// TIA Portal V18 export
FUNCTION_BLOCK "Conveyor"   // FB2, FBD
{ S7_Optimized_Access := 'TRUE' }
VERSION : 0.1
// stored: AutoNumber true, IsIECCheckEnabled true, IsRetainMemResEnabled false, MemoryReserve 100, SetENOAutomatically false, UDAEnableTagReadback false
   VAR_INPUT
      automaticMode : Bool;
      manualMode : Bool;
      jogRight : Bool;
      run : Bool;
   END_VAR
   VAR_OUTPUT
      conveyorRight : Bool;
      conveyorLeft : Bool;
   END_VAR
   VAR
      statRequest : Bool;
      statRelease : Bool;
   END_VAR
BEGIN

REGION Network 1 (SCL)
   //=============================================================================
   //Siemens AG // (c)Copyright (2018)
   //-----------------------------------------------------------------------------
   // Library: -
   // Tested with: CPU 1517-3 PN/DP V2.5
   // Engineering: TIA Portal V15
   // Restrictions: -
   // Requirements: PLC (S7-1500)
   // Functionality: Conveyor
   //-----------------------------------------------------------------------------
   // Change log table:
   // Version  Date      Expert in charge  Changes applied
   // 01.00.00 24.08.18  Siemens           First released version
   //=============================================================================
END_REGION

REGION Network 2
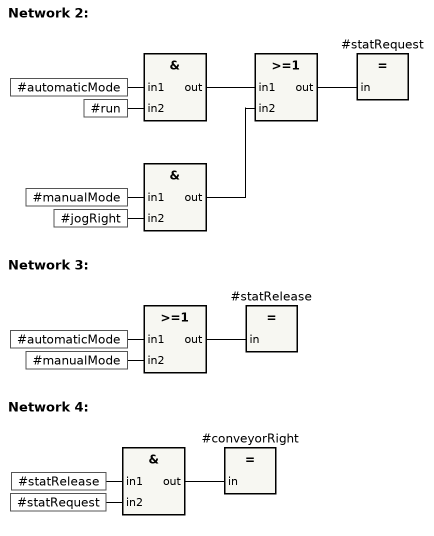
   #statRequest := (#automaticMode AND #run) OR (#manualMode AND #jogRight);
END_REGION

REGION Network 3
   #statRelease := #automaticMode OR #manualMode;
END_REGION

REGION Network 4
   #conveyorRight := #statRelease AND #statRequest;
END_REGION
END_FUNCTION_BLOCK
